FUNCTION Execute_Write_Screen : BOOL
VAR_INPUT
END_VAR
VAR
END_VAR

GV_MODBUS.addr := GV_MODBUS.oneLeftAddr;
GV_MODBUS.writeExecute := TRUE;
GV_MODBUS.readExecute := FALSE;
GV_MODBUS.doneWriting := FALSE;
GV_MODBUS.btnData := 0;

END_FUNCTION

(* stored: Version 1.1.0.1, ProductVersion 3.1.4022.12
   POU Execute_Write_Screen: Id {c34f2788-754d-42b5-a5c7-b5a1c4b4c671}, SpecialFunc None *)
